(* PLC project Unnamed, Неизвестно Unnamed 1 *)
(* stored: creationDateTime 2024-04-02T10:29:43, modificationDateTime 2025-02-03T01:14:21 *)

PROGRAM OvenPCB
  VAR
    mb_PWM_freq_h AT %QW100 : INT;
    mb_PWM_freq_l AT %QW101 : INT;
    mb_PWM_duty AT %QW102 : INT;
    mb_Temp AT %IW100 : INT;
    mb_TempDS18B20 AT %IW101 : INT;
    mbsl_Temp AT %QW0 : INT;
    mbsl_TempDS18B20 AT %QW1 : INT;
  END_VAR
  VAR
    PID0 : PID;
  END_VAR
  VAR
    PID_Auto AT %QX0.0 : BOOL := FALSE;
    PID_Out AT %MD0 : REAL;
    PID_P AT %MD1 : REAL := 2.0;
    PID_I AT %MD2 : REAL := 1000.0;
    PID_D AT %MD3 : REAL := 0.0;
    PID_SP AT %MD4 : REAL := 450.0;
    PWM_duty AT %MD5 : DINT;
    PWM_duty_manual AT %MD6 : REAL := 0.0;
  END_VAR
  VAR  (* added by the conversion: wires and edge detectors of the diagram *)
    _SUB65_OUT : INT;
    _LIMIT60_OUT : INT;
  END_VAR

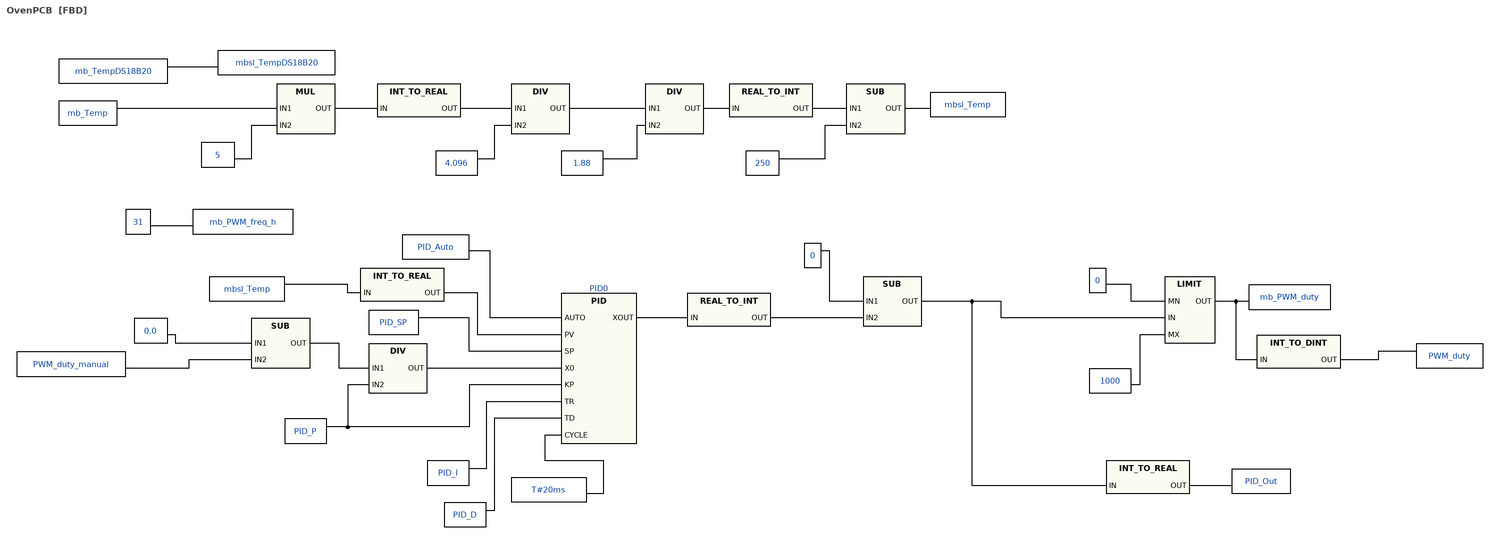
(* FBD diagram, written out as Structured Text *)
PID0(AUTO := PID_Auto, PV := INT_TO_REAL(mbsl_Temp), SP := PID_SP, X0 := (0.0 - PWM_duty_manual) / PID_P, KP := PID_P, TR := PID_I, TD := PID_D, CYCLE := T#20ms);
_SUB65_OUT := 0 - REAL_TO_INT(PID0.XOUT);
_LIMIT60_OUT := LIMIT(0, _SUB65_OUT, 1000);
mb_PWM_duty := _LIMIT60_OUT;
mb_PWM_freq_h := 31;
mbsl_Temp := REAL_TO_INT(INT_TO_REAL(mb_Temp * 5) / 4.096 / 1.88) - 250;
mbsl_TempDS18B20 := mb_TempDS18B20;
PID_Out := INT_TO_REAL(_SUB65_OUT);
PWM_duty := INT_TO_DINT(_LIMIT60_OUT);
END_PROGRAM

CONFIGURATION Config0
  RESOURCE Res0 ON PLC
    TASK task0(INTERVAL := T#20ms, PRIORITY := 0);
    PROGRAM instance0 WITH task0 : OvenPCB;
  END_RESOURCE
END_CONFIGURATION
